PROGRAM MAIN
VAR
	fbStateMachinePro : FB_StateMachinePro;
END_VAR

fbStateMachinePro(
	bEnable:= TRUE, 
	bStart:= GVL.bStart, 
	bStop:= GVL.bStop, 
	bBottle:= GVL.bBottle, 
);

GVL.bConveyor := fbStateMachinePro.bConveyor;
GVL.bWater := fbStateMachinePro.bWater;
GVL.bMint := fbStateMachinePro.bMint;	
GVL.bCorking := fbStateMachinePro.bCorking;

END_PROGRAM

(* stored: Version 1.1.0.1, ProductVersion 3.1.4024.12
   POU MAIN: Id {41c4aa59-1c6a-4a73-9d14-43b9b6d789a2}, SpecialFunc None *)
